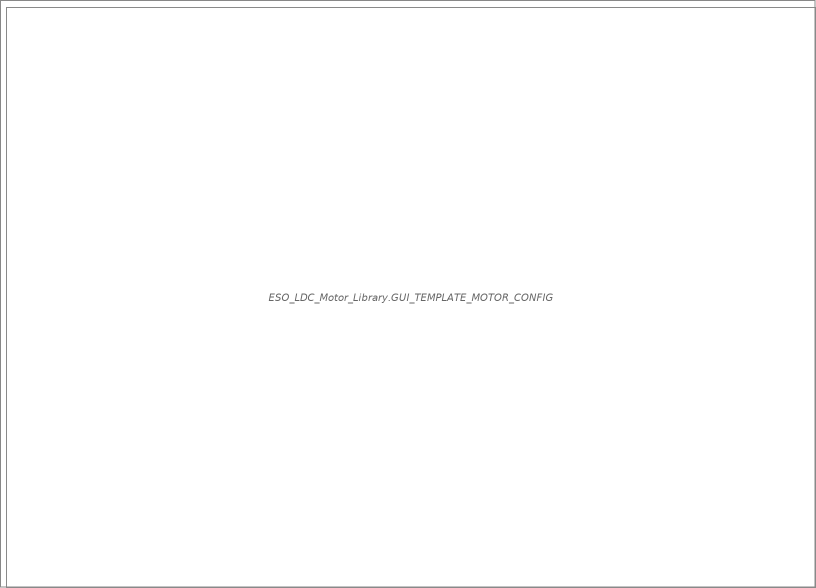
VISUALIZATION Motor001_Config  // 816x588
    Frame (6,7 810x581)
        shows ESO_LDC_Motor_Library.GUI_TEMPLATE_MOTOR_CONFIG(m_Instance := MAIN.Motor001)
END_VISUALIZATION

(* stored: Version 1.1.0.1, ProductVersion 3.1.4024.9
   Visu Motor001_Config: Id {d173b763-f032-490a-bfdf-03d7cf0127fc} *)
